Fanuc KAREL source: ka00066.KL

-- PROVISIONAL review KL for V770-1; original PC SHA256 801cd7a80e80925941b402eb713d26660403d9db6af808c0d2fe31d86de12528
-- Incomplete behavior may be omitted. Consult companion uncertainty JSON. Do not deploy.
PROGRAM KA00066
%NOLOCKGROUP
-- UNRESOLVED_DECL SRC type=000102
-- UNRESOLVED_DECL DST type=000102
BEGIN
  -- UNRESOLVED_PC offsets 5-20; opcodes 2E,22,32,35
  -- UNRESOLVED_PC offsets 25-40; opcodes 49,4A
  -- UNRESOLVED_PC offsets 45-49; opcodes 7F
END KA00066
